INTERFACE I_PackML_Mode

METHOD PUBLIC Abort
VAR_INPUT
END_VAR
END_METHOD

METHOD PUBLIC Clear
VAR_INPUT
END_VAR
END_METHOD

PROPERTY PUBLIC CurrentState : PackML_State
GET
END_GET
END_PROPERTY

METHOD PUBLIC CyclicCall
VAR_INPUT
END_VAR
END_METHOD

METHOD PUBLIC Hold
VAR_INPUT
END_VAR
END_METHOD

PROPERTY PUBLIC IsAborted : bool
GET
END_GET
END_PROPERTY

PROPERTY PUBLIC IsAborting : bool
GET
END_GET
END_PROPERTY

PROPERTY PUBLIC IsClearing : bool
GET
END_GET
END_PROPERTY

PROPERTY PUBLIC IsComplete : bool
GET
END_GET
END_PROPERTY

PROPERTY PUBLIC IsCompleting : bool
GET
END_GET
END_PROPERTY

PROPERTY PUBLIC IsExecuting : bool
GET
END_GET
END_PROPERTY

PROPERTY PUBLIC IsHeld : bool
GET
END_GET
END_PROPERTY

PROPERTY PUBLIC IsHolding : bool
GET
END_GET
END_PROPERTY

PROPERTY PUBLIC IsIdle : BOOL
GET
END_GET
END_PROPERTY

METHOD PUBLIC IsModeTransitionAllowed : BOOL
VAR_INPUT
	
END_VAR
END_METHOD

PROPERTY PUBLIC IsResetting : bool
GET
END_GET
END_PROPERTY

PROPERTY PUBLIC IsStarting : bool
GET
END_GET
END_PROPERTY

PROPERTY PUBLIC IsStopped : BOOL
GET
END_GET
END_PROPERTY

PROPERTY PUBLIC IsStopping : bool
GET
END_GET
END_PROPERTY

PROPERTY PUBLIC IsSuspended : bool
GET
END_GET
END_PROPERTY

PROPERTY PUBLIC IsSuspending : bool
GET
END_GET
END_PROPERTY

PROPERTY PUBLIC IsUnholding : bool
GET
END_GET
END_PROPERTY

PROPERTY PUBLIC IsUnsuspending : bool
GET
END_GET
END_PROPERTY

METHOD PUBLIC Reset
VAR_INPUT
END_VAR
END_METHOD

METHOD PUBLIC Start
VAR_INPUT
END_VAR
END_METHOD

METHOD PUBLIC Stop
VAR_INPUT
END_VAR
END_METHOD

METHOD PUBLIC Suspend
VAR_INPUT
END_VAR
END_METHOD

METHOD PUBLIC Unhold
VAR_INPUT
END_VAR
END_METHOD

METHOD PUBLIC Unsuspend
VAR_INPUT
END_VAR
END_METHOD

END_INTERFACE

(* stored: Version 1.1.0.1, ProductVersion 3.1.4024.12
   Itf I_PackML_Mode: Id {97fc6d2f-c469-4986-a6ff-20099b2007b5}
   Folder Properties: Id {cb4b7309-a058-470e-aac8-fac2e1e7c07f}
   Folder Public: Id {f3cdd0d6-b9cd-4fbc-be23-18918415331b}
   Method Abort: Id {d65dcde3-6a3b-4d68-92ca-d7db64a16943}
   Method Clear: Id {50999d02-ae62-45b8-b7bd-001050f2aab4}
   Property CurrentState: Id {654531f9-76ae-4aef-8560-1c397ee53157}
   Get Get: Id {ce8e1346-6609-41ed-b00d-dc8c4571d758}
   Method CyclicCall: Id {d5bbdca6-03e6-4649-ae79-8146379d0d79}
   Method Hold: Id {612804b0-88e8-444e-b1c2-038d511f2570}
   Property IsAborted: Id {0f9d10af-1131-4b57-94d1-21a74074f8a0}
   Get Get: Id {45b6c7b4-0738-45a0-8f9c-8f109116aee6}
   Property IsAborting: Id {fda16094-c26e-4c85-854f-9b5fc3c5e219}
   Get Get: Id {a750d063-1893-4ff3-a543-97fc3d3db347}
   Property IsClearing: Id {77435faf-9e4f-4c13-9d44-30be9e7fa103}
   Get Get: Id {f74f08e5-2b88-49c7-a882-82c6db3ca8c1}
   Property IsComplete: Id {178be6a9-d50b-4d65-bbb2-2cf7c1409d95}
   Get Get: Id {1342af11-f084-4991-836c-dfc0f7215918}
   Property IsCompleting: Id {dfbf910e-7c4c-47ea-a1fb-03bc48272f3f}
   Get Get: Id {c249a34e-332d-4258-b068-47a3b4805971}
   Property IsExecuting: Id {86d16397-2c29-4600-9416-38af4206106e}
   Get Get: Id {d5bfe5f7-5fd9-4a20-b677-d27d3fc54666}
   Property IsHeld: Id {d4c55b30-1f4c-4974-a84f-01dc15533072}
   Get Get: Id {7f692ea5-01d6-4285-bfbc-2957ac45c82f}
   Property IsHolding: Id {5cb0ab24-73b5-48d1-8057-2746e68a66b8}
   Get Get: Id {2ebc6ebb-5f62-4d45-877f-f640ee3869a4}
   Property IsIdle: Id {544f8f54-c54a-488e-b1b2-86544b9f41c7}
   Get Get: Id {7177968b-d3f7-4aac-9549-652cae29f743}
   Method IsModeTransitionAllowed: Id {7275b0f2-063d-4ab7-94fb-0d991fa87e5d}
   Property IsResetting: Id {ab94db72-b0d9-4038-b4fc-21d3d063426d}
   Get Get: Id {39a417af-ba5b-4ee9-bb0d-4dc0ce5c9ee1}
   Property IsStarting: Id {0d5b39dd-aad0-4cf2-9e5c-5b535305f105}
   Get Get: Id {20eb0ad7-36f5-46ae-b5b8-e4c82f881c7b}
   Property IsStopped: Id {a0337ac8-f0a5-400b-80d3-8ffb8259350c}
   Get Get: Id {a5caafea-7157-460c-aae1-36b5e4ff08d3}
   Property IsStopping: Id {7867ddbe-8832-4abe-b670-959ff6cbbe15}
   Get Get: Id {d8b8aea0-6ab5-42aa-8986-dfff3dbaa305}
   Property IsSuspended: Id {0c9795dd-5ffe-4317-add5-84dc288635f9}
   Get Get: Id {7e9bbbac-2bf8-4e8b-a2dd-4a44bfdc330c}
   Property IsSuspending: Id {fd0fefd1-fec5-4681-a0ee-123763602fe1}
   Get Get: Id {7f2432b6-bd28-46f8-8024-156d2719bb9f}
   Property IsUnholding: Id {1b9a5b88-f010-4dc9-aa64-064bd11dc99c}
   Get Get: Id {45e2f4ef-521b-4f4c-886a-f35a7ec7e630}
   Property IsUnsuspending: Id {a3030584-e1a8-48d1-8a81-0e91921a8325}
   Get Get: Id {7b27baac-4724-4324-9501-f39a3c2fcd45}
   Method Reset: Id {12eb6aea-34fa-423d-96a6-f375ac6163ff}
   Method Start: Id {1c086114-3605-4910-9e0a-9b8187d5c8a8}
   Method Stop: Id {669e7c7a-38f8-4c04-a257-a9705a029e82}
   Method Suspend: Id {c197dd01-36c6-44c4-9ecc-a65c3b56b859}
   Method Unhold: Id {b66587e4-567a-455a-b116-8e51385e6b2c}
   Method Unsuspend: Id {02f2747e-de47-434d-a076-a04bab3b5e8e} *)
